TYPE ST_SafetyFunction :
STRUCT
    refSafetyIn : REFERENCE TO ST_SafetyFunctionIn;
    refSafetyOut : REFERENCE TO ST_SafetyFunctionOut;
END_STRUCT
END_TYPE

(* stored: Version 1.1.0.1
   DUT ST_SafetyFunction: Id {58782b85-35f4-479a-95a9-2262a8ca7afe} *)
